FUNCTION_BLOCK STARTER_BUTTON (* Start Interface *)
  (* Standard: 61499-2 *)
  (* Version BETA, 17/01/2012, Universidade do Estado de Santa Catarina *)
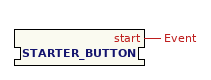
  EVENT_OUTPUT
    start;
  END_EVENT
  SERVICE USER/STARTER (* Starter Service *)
    SEQUENCE START
      USER.USER() -> STARTER_BUTTON.start();
    END_SEQUENCE
  END_SERVICE
END_FUNCTION_BLOCK
